Yaskawa INFORM job: X2_50&56A(90,0).JBI

/JOB
//NAME X2_50&56A(90,0)
//POS
///NPOS 390,390,390,18,0,0
///TOOL 0
///POSTYPE PULSE
///PULSE
C00000=-35013,-75230,-81678,-29902,96544,59223
C00001=-146238,44864,29954,-30461,95448,60806
C00002=-147931,42899,30637,-30414,93594,60637
C00003=-149034,42975,32803,-30382,92069,60611
C00004=-149034,43187,33728,-30365,91671,60717
C00005=-148618,42187,30995,-30400,92836,60570
C00006=-146730,40288,31403,-30303,92453,61410
C00007=-147687,41392,32561,-30326,91981,61161
C00008=-146730,40288,31403,-30303,92453,61410
C00009=-146628,38101,29073,-30312,92759,61369
C00010=-146969,35065,25949,-30338,92951,61185
C00011=-146628,38101,29073,-30312,92759,61369
C00012=-145936,38825,28710,-30317,93527,61436
C00013=-144232,40818,28013,-30345,95405,61605
C00014=-133297,17715,2025,-3580,100928,70099
C00015=-121777,-29733,-12388,29914,87306,80525
C00016=-120032,-31040,-9886,30121,84762,80532
C00017=-119311,-31474,-8810,30220,83736,80539
C00018=-119316,-30440,-7071,30243,83270,80413
C00019=-119316,-29997,-6042,30262,82917,80320
C00020=-120906,-31495,-8824,30067,84297,80075
C00021=-122289,-30144,-5697,29969,83711,79393
C00022=-122317,-32815,-7460,29979,83470,79319
C00023=-122289,-30144,-5697,29969,83711,79393
C00024=-122735,-29704,-5039,29928,83710,79223
C00025=-121134,-29738,-5062,30101,83147,79686
C00026=-122735,-29704,-5039,29928,83710,79223
C00027=-126540,-28280,-10143,29422,88423,78984
C00028=-68546,9416,10683,17932,104217,63227
C00029=-68516,6763,11888,17759,102202,62934
C00030=-68503,6025,13208,17671,101063,62768
C00031=-68451,6691,14972,17632,100341,62681
C00032=-68503,5773,12452,17696,101383,62816
C00033=-66565,12547,20523,18047,99542,63243
C00034=-65781,10285,18484,18233,99456,63513
C00035=-66565,12547,20523,18047,99542,63243
C00036=-65967,10809,19346,18174,99249,63415
C00037=-66882,8922,17759,17963,99458,63116
C00038=-65967,10809,19346,18174,99249,63415
C00039=-66084,14240,17447,18358,102066,63804
C00040=-115698,-30544,-51433,15731,84190,63390
C00041=-118338,-32636,-46922,7735,73478,10834
C00042=-114067,48339,9442,8727,107260,-37267
C00043=-101651,53791,20065,8419,102302,-33380
C00044=-100782,53794,25900,8285,98661,-33332
C00045=-100318,54126,27705,8251,97683,-33240
C00046=-100315,54082,28901,8233,96933,-33289
C00047=-100318,54126,27705,8251,97683,-33240
C00048=-103340,51772,25926,13303,96601,-33902
C00049=-102638,52333,26542,13275,96399,-33681
C00050=-103340,51772,25926,13303,96601,-33902
C00051=-103881,51441,24204,13355,97556,-33985
C00052=-105240,51372,17279,13610,101889,-33974
C00053=-105263,53169,23809,16124,107359,-67725
C00054=-105263,53098,24698,16066,106796,-67804
C00055=-105263,53109,24538,16076,106896,-67790
C00056=-105080,50164,21304,16137,107318,-67665
C00057=-105202,52155,23020,16124,107309,-67712
C00058=-106286,50684,21405,16057,107747,-68046
C00059=-106213,46871,17829,16087,107966,-67990
C00060=-105813,47115,18093,16117,107853,-67859
C00061=-106213,47152,15738,16242,109344,-67797
C00062=-102863,-18246,-47623,4026,92422,-23125
C00063=-102376,-34818,-59840,10840,84298,-4292
C00064=-100002,-32974,-49147,13806,76787,-3743
C00065=-100270,-30914,-48271,13869,77337,-3774
C00066=-100148,-31724,-49706,13807,77772,-3684
C00067=-99723,-30030,-48565,13661,77867,-3527
C00068=-99723,-30105,-48044,13677,77517,-3566
C00069=-99495,-31680,-49824,13589,77759,-3462
C00070=-97800,-40718,-55675,5005,73967,4597
C00071=-93318,-38382,-52327,94,72702,9054
C00072=-92851,-38032,-52104,-83,72745,9214
C00073=-95045,-39040,-57560,738,75594,8477
C00074=-124861,-15271,-40833,8838,93503,-41842
C00075=-136908,-36114,-55425,10666,93196,-45849
C00076=-135773,-37299,-49208,10462,88689,-45850
C00077=-136921,-36837,-46377,10628,87355,-46351
C00078=-136921,-36755,-44333,10633,86159,-46454
C00079=-136921,-36814,-45592,10627,86891,-46392
C00080=-117319,-40034,-47848,-16199,85186,-41646
C00081=-117335,-39772,-46156,-16213,84312,-41538
C00082=-116208,-39661,-46084,-16390,84550,-41175
C00083=-118605,-39981,-48556,-15987,85383,-42119
C00084=-142194,-34441,-52424,11225,92893,-47663
C00085=-137296,-41112,-44413,7882,96909,-45970
C00086=-121079,-43154,-38901,8183,90890,-40792
C00087=-119046,-42134,-34632,8196,88600,-40245
C00088=-118232,-41637,-32862,8204,87692,-40026
C00089=-118232,-41216,-31330,8206,86972,-40073
C00090=-118232,-41637,-32862,8204,87692,-40026
C00091=-123515,-41178,-31164,13251,87604,-41880
C00092=-122294,-41232,-31198,13272,87397,-41478
C00093=-123515,-41178,-31164,13251,87604,-41880
C00094=-124446,-41576,-32799,13232,88537,-42104
C00095=-126767,-42340,-36726,13193,90889,-42661
C00096=-121202,-54016,-38461,8184,85107,-41211
C00097=-118951,-52355,-33810,8234,82889,-40587
C00098=-118051,-51605,-31888,8256,82008,-40337
C00099=-118051,-50970,-30224,8268,81318,-40383
C00100=-118051,-51605,-31888,8256,82008,-40337
C00101=-123729,-51057,-30474,13322,82279,-42525
C00102=-122379,-51113,-30506,13351,82049,-42081
C00103=-123729,-51057,-30474,13322,82279,-42525
C00104=-120943,-27615,-16514,12405,97908,-68352
C00105=-120948,-30071,-17086,12372,97018,-68441
C00106=-120951,-31730,-18195,12366,96852,-68459
C00107=-120948,-30071,-17086,12372,97018,-68441
C00108=-124760,-51678,-32249,13279,83200,-42783
C00109=-127326,-53005,-36529,13179,85520,-43425
C00110=-154326,-120554,-77654,11334,79888,-63138
C00111=-167720,-105639,-119673,16034,110248,-69380
C00112=-180425,17295,-38776,18903,121217,-77748
C00113=-160704,-72602,-79591,10350,105538,-81389
C00114=-159985,-76902,-77997,10237,102306,-81413
C00115=-158839,-75685,-75597,10284,101324,-81094
C00116=-158717,-75119,-73898,10260,100564,-81114
C00117=-159022,-76399,-75134,10243,100704,-81209
C00118=-159327,-81052,-76621,10164,99289,-81434
C00119=-159429,-77687,-75590,10198,100380,-81379
C00120=-160454,-72036,-78000,10329,104829,-81362
C00121=-122590,-90956,-95479,-6285,107811,-74232
C00122=-122432,-96187,-93928,-6136,104200,-73988
C00123=-122366,-98076,-93201,-6086,102795,-73894
C00124=-122349,-96392,-90986,-6070,102302,-73864
C00125=-122333,-96702,-91360,-6071,102373,-73862
C00126=-121172,-100063,-92157,-5915,101229,-73400
C00127=-122333,-96702,-91360,-6071,102373,-73862
C00128=-116908,-96303,-91435,-5489,103011,-71994
C00129=-118888,-98383,-91954,-5688,102128,-72646
C00130=-116908,-96303,-91435,-5489,103011,-71994
C00131=-117392,-89431,-93773,-5700,107925,-72394
C00132=-123779,-92334,-96085,11860,100478,-68930
C00133=-121799,-96099,-93963,11739,97018,-68578
C00134=-121068,-94931,-92225,11724,96454,-68379
C00135=-120976,-95732,-90808,11689,95182,-68467
C00136=-121047,-96000,-91535,11697,95495,-68462
C00137=-119860,-99344,-92335,11668,94123,-68181
C00138=-121047,-96000,-91535,11697,95495,-68462
C00139=-119543,-98346,-92112,11677,94445,-68041
C00140=-121592,-100306,-92571,11657,94029,-68789
C00141=-119543,-98346,-92112,11677,94445,-68041
C00142=-122418,-93690,-95360,11815,99162,-68586
C00143=-124052,-92327,-98574,11935,102020,-68874
C00144=-122075,-96496,-96608,11789,98453,-68536
C00145=-121256,-97943,-95721,11744,97072,-68385
C00146=-121250,-96320,-93531,11728,96567,-68431
C00147=-121163,-96877,-94234,11732,96698,-68388
C00148=-119974,-100369,-95083,11696,95280,-68111
C00149=-121163,-96877,-94234,11732,96698,-68388
C00150=-120506,-98881,-94746,11711,95903,-68236
C00151=-118500,-96784,-94222,11730,96355,-67499
C00152=-120506,-98881,-94746,11711,95903,-68236
C00153=-123349,-93657,-97773,11879,100767,-68753
C00154=-135291,-86613,-75974,52977,86020,-81582
C00155=-131116,-88371,-74218,52881,82397,-81428
C00156=-129398,-88910,-73439,52861,80942,-81342
C00157=-128447,-91701,-74067,52932,79748,-81525
C00158=-130431,-95374,-76659,53055,80707,-82053
C00159=-128834,-93195,-74891,52983,79809,-81703
C00160=-130431,-95374,-76659,53055,80707,-82053
C00161=-124555,-94103,-78793,52446,78563,-80078
C00162=-125999,-93781,-77341,52659,78933,-80655
C00163=-124555,-94103,-78793,52446,78563,-80078
C00164=-130787,-92210,-81525,52671,83776,-80437
C00165=-125882,-96985,-97972,20817,92084,-56602
C00166=-122325,-98161,-95172,20440,89016,-55857
C00167=-120880,-94284,-92066,20293,88735,-55390
C00168=-120880,-94153,-90803,20292,88068,-55501
C00169=-120880,-94284,-92066,20293,88735,-55390
C00170=-119026,-94251,-92054,20095,88291,-54803
C00171=-120880,-94284,-92066,20293,88735,-55390
C00172=-120884,-98206,-92897,20294,87320,-55628
C00173=-120880,-94284,-92066,20293,88735,-55390
C00174=-125854,-95536,-95978,20803,91624,-56671
C00175=-125850,-66912,-79659,30836,57983,-58657
C00176=-122561,-63207,-75462,29110,56252,-57732
C00177=-121295,-61670,-73737,28426,55590,-57365
C00178=-121291,-60661,-71640,28674,54906,-57565
C00179=-121285,-60765,-71809,28654,54949,-57550
C00180=-119473,-60737,-71796,27523,54360,-56906
C00181=-121285,-60765,-71809,28654,54949,-57550
C00182=-119935,-60692,-71734,27818,54496,-57075
C00183=-119959,-57359,-70502,27528,55354,-56840
C00184=-119935,-60692,-71734,27818,54496,-57075
C00185=-124401,-66105,-77764,30230,56821,-58377
C00186=-128142,-64639,-90036,18676,74706,-62694
C00187=-138485,-71827,-101197,-11106,105399,-77644
C00188=-147024,-87385,-83593,-35439,109592,-87133
C00189=-149732,-92665,-83137,-35225,106008,-87097
C00190=-150982,-92517,-82536,-35527,105093,-87095
C00191=-150854,-90774,-79322,-35312,104257,-86759
C00192=-145431,-93697,-76928,-39294,101207,-75263
C00193=-143884,-94649,-78323,-39224,102144,-74704
C00194=-141496,-90316,-79520,-39399,105550,-74933
C00195=-154875,-73459,-94031,3699,115712,-75473
C00196=-154642,-88430,-80864,46638,100530,-71967
C00197=-150685,-92332,-80273,46535,96810,-71811
C00198=-149068,-93915,-80023,46523,95290,-71747
C00199=-152233,-91403,-76041,46197,96115,-72893
C00200=-138023,-100193,-87798,32403,89280,-71025
C00201=-139486,-99224,-88637,32451,90704,-71199
C00202=-143008,-96307,-90518,32622,94313,-71562
C00203=-126401,-92982,-99947,26116,71912,-46119
C00204=-122401,-89174,-95921,24616,70248,-44972
C00205=-121170,-87691,-94393,24143,69731,-44617
C00206=-121073,-40431,-77118,23973,104037,-41292
C00207=-121948,-141376,-105315,24084,72465,-47862
C00208=-119793,-124223,-100539,21665,86903,-40754
C00209=-121070,-126388,-102412,21638,87354,-41108
C00210=-126026,-127807,-105919,21532,89991,-42436
C00211=-136654,-67846,-101646,-5444,103045,-74682
C00212=-128322,-96725,-99076,14451,99613,-67284
C00213=-128011,-95143,-96681,14417,98917,-67259
C00214=-125059,-98267,-95078,14269,95825,-66574
C00215=-132883,-103944,-96240,14189,95056,-69399
C00216=-122114,-97273,-96139,7492,99903,-69823
C00217=-123656,-92823,-98050,7552,103478,-70135
C00218=-148370,-106244,-91268,32547,97235,-62203
C00219=-143957,-109023,-89633,32719,93465,-61524
C00220=-142187,-110300,-89017,32799,91899,-61269
C00221=-110014,-102343,-95219,10833,94604,-66470
C00222=-122878,-112804,-97097,10537,93258,-71032
C00223=-110561,-104342,-93907,1603,99479,-78541
C00224=-110841,-84726,-85708,1760,111290,-78449
C00225=-111201,-78802,-86432,1737,114786,-78527
C00226=-106717,-60158,-79706,8194,107324,-64031
C00227=-105123,-63987,-78019,8070,104193,-63696
C00228=-104341,-64830,-77125,8038,103145,-63496
C00229=-106614,-68907,-78610,7970,102193,-64341
C00230=-164586,-101102,-83968,4841,93825,-84736
C00231=-168005,-100380,-83271,4564,93970,-85900
C00232=-165984,-96075,-92358,4843,101626,-84914
C00233=-181857,-131319,-116911,12842,90499,-90722
C00234=-202989,-63880,-99903,47799,99542,-84030
C00235=-168472,-147890,-132681,14947,97151,-71352
C00236=-154326,-120554,-77654,11334,79888,-63138
C00237=-128098,-77833,-51544,-1657,63239,-16727
C00238=-116532,-49017,-34945,-4360,90951,-81305
C00239=-116532,-49017,-34945,-4360,90951,-81305
C00240=-116798,-50663,-32111,-4378,88355,-81305
C00241=-116908,-51227,-30905,-4388,87320,-81307
C00242=-119609,-51392,-30999,-4620,87132,-82211
C00243=-121719,-51405,-31006,-4797,87008,-82917
C00244=-124421,-51272,-30929,-5019,86875,-83824
C00245=-124228,-50732,-32149,-5002,87911,-83800
C00246=-145745,-14259,570,10366,107018,-74117
C00247=-149880,-18384,-846,13396,104500,-71178
C00248=-151111,-18464,18,13945,103653,-70648
C00249=-151285,-17723,1623,13844,103092,-70775
C00250=-151490,-18588,-4768,14034,106516,-70446
C00251=-99208,-22167,-7317,-16130,105202,-90552
C00252=-102111,-21459,-2862,-15110,103391,-89386
C00253=-101894,-21074,-1790,-15006,102986,-89257
C00254=-101783,-20670,-1192,-14957,102851,-89201
C00255=-100868,-20755,-6903,-14931,106373,-89315
C00256=-123764,-49143,-35016,-4968,90511,-83746
C00257=-123498,-46334,-32145,14225,106729,-81506
C00258=-122671,-49917,-31274,14287,104276,-81501
C00259=-122321,-51270,-30849,14324,103286,-81493
C00260=-121710,-51281,-30881,14509,103202,-81284
C00261=-119621,-51322,-31009,15133,102879,-80573
C00262=-119011,-51335,-31052,15312,102775,-80367
C00263=-119414,-50002,-31488,15265,103772,-80384
C00264=-116044,-49795,-31370,16241,103155,-79243
C00265=-112158,-52942,-30337,13826,98266,-82965
C00266=-122910,-69671,-38655,20695,87695,-72461
C00267=-124804,-70759,-45426,20434,91550,-72479
C00268=-120368,-46468,-32388,15179,106240,-80415
C00269=-103583,-18395,-21065,18333,98049,-47386
C00270=-95522,-2033,346,19157,86542,-33647
C00271=-95065,-1179,4289,19188,84551,-33796
C00272=-94194,-282,6213,19202,83664,-33623
C00273=-92524,-10041,-1636,19198,83097,-33115
C00274=-94699,28090,37444,23065,99649,-38348
C00275=-95245,43682,55653,23027,103524,-40317
C00276=-97031,45002,54317,22569,105398,-40615
C00277=-95302,21282,15864,17128,100326,-40606
C00278=-95633,-1961,-1285,16168,78923,-31701
C00279=-94125,315,3726,16087,76781,-31446
C00280=-93197,3589,10969,16156,73926,-31495
C00281=-93115,4380,12654,16195,73301,-31552
C00282=-94556,14113,21261,16393,73308,-32073
C00283=-94819,12763,18273,16338,74461,-32010
C00284=-94855,11979,15831,16266,75524,-31879
C00285=-94760,268,4885,16208,76196,-31753
C00286=-93262,3253,10079,16136,74301,-31466
C00287=-93099,4430,12776,16195,73253,-31551
C00288=-94504,14241,21527,16396,73200,-32069
C00289=-94774,13150,19338,16366,74011,-32057
C00290=-95480,10422,13554,16303,76229,-32007
C00291=-97216,11756,13085,16445,77515,-32459
C00292=-95984,14761,19072,16436,75210,-32328
C00293=-95926,15643,20974,16479,74507,-32404
C00294=-96702,21319,26244,16596,74351,-32707
C00295=-88276,-5311,8070,1704,50857,-22867
C00296=-87929,-9523,3732,1524,51354,-22713
C00297=-88057,-15039,-3820,1549,53169,-22739
C00298=-99387,-43194,-40222,6284,61646,-26942
C00299=-121163,30977,-5145,19643,99311,-32181
C00300=-111536,75135,35465,20047,103602,-28019
C00301=-109733,75701,42270,19665,99503,-28062
C00302=-107396,77633,44085,15199,99812,-27662
C00303=-106846,74881,40767,13783,95666,-18812
C00304=-105506,42598,5344,10183,85057,-21764
C00305=-107494,36842,-4476,11925,85901,-22339
C00306=-110038,51949,7342,17956,100045,-24263
C00307=-110492,43774,10982,19918,106123,-35860
C00308=-109482,36992,6821,19832,105013,-35683
C00309=-108373,36531,10179,19621,102581,-35693
C00310=-107789,34301,9135,19587,101968,-35584
C00311=-105866,51618,28942,18605,112563,-37835
C00312=-106064,56056,31872,17240,113701,-37835
C00313=-105930,58571,31891,15493,114477,-37831
C00314=-113418,37409,2332,24084,99798,-37219
C00315=-113418,37409,2332,24084,105102,-80908
C00316=-113160,50873,23237,25434,107555,-80153
C00317=-112025,51272,23640,25519,107174,-79798
C00318=-112126,54336,25481,25581,107605,-79738
C00319=-108217,56173,27527,25805,106134,-78563
C00320=-108012,53365,25864,25757,105690,-78586
C00321=-107358,53539,26056,25793,105464,-78385
C00322=-107594,58308,28543,25913,106367,-78268
C00323=-114507,53473,22978,25568,109314,-80271
C00324=-122054,65837,41057,36395,121722,-57977
C00325=-123579,42738,19822,41051,112959,-51179
C00326=-124152,34164,13148,42323,109003,-48943
C00327=-124227,34353,16593,41799,107514,-49624
C00328=-126462,36438,15351,42046,109959,-49631
C00329=-128176,29859,1512,43519,114603,-48350
C00330=-130467,-18606,-44219,44095,94408,31747
C00331=-121945,-44389,-49110,46115,69080,26022
C00332=-121904,-40131,-44420,46290,68567,25788
C00333=-113124,-39530,-44042,43500,64204,28113
C00334=-112945,-43259,-50161,42865,65486,28791
C00335=-113288,-45265,-40830,46737,56763,24195
C00336=-111978,-45017,-40682,46242,56106,24578
C00337=-111880,-47039,-43845,45778,56697,24958
C00338=-122010,-47932,-44372,49222,61967,22192
C00339=-118733,-49642,-44567,45028,57156,26003
C00340=-115692,-49409,-44472,43850,55672,26913
C00341=-119979,-54076,-53442,44153,60090,26830
C00342=-127641,-46610,-57429,46858,74797,25997
C00343=-135004,-69306,-84470,28637,83306,-48309
C00344=-114761,-54427,-46396,25764,86438,-35617
C00345=-80124,-32108,-24664,-24795,97657,55749
C00346=-97606,39512,4524,-30816,78189,70702
C00347=-104188,47256,24507,-29638,68650,70716
C00348=-105086,62165,41181,-29824,66062,71062
C00349=-101009,53751,26030,-30366,71859,71113
C00350=-95324,41094,10845,-31949,76382,71947
C00351=-87558,21315,-14177,-31275,118027,78587
C00352=-99257,8968,-10542,-28789,118245,76702
C00353=-100154,5822,-7742,-28106,114988,77225
C00354=-99796,6145,-6533,-27877,114593,77484
C00355=-99255,6664,-4734,-27546,114022,77862
C00356=-106453,5544,-9246,-16915,113806,78351
C00357=-106832,8673,-12915,-17628,117423,77625
C00358=-94457,17302,-8508,-14643,121478,81992
C00359=-77268,892,-37386,-36976,90749,74597
C00360=-55933,-105254,-98782,-41109,86932,84870
C00361=-92475,-165326,-103936,3399,48061,-39515
C00362=-111759,-161502,-101201,19707,45151,-81968
C00363=-123409,-143891,-91937,22487,51121,-85856
C00364=-115094,-142630,-90727,15919,48927,-82057
C00365=-105882,-142342,-91359,8372,48357,-77561
C00366=-52718,-102797,-81138,-14928,68501,-56921
C00367=-53797,-105289,-84123,-14624,68845,-57366
C00368=-54179,-107975,-89277,-14378,70514,-57714
C00369=-16825,-139657,-107848,-21320,74237,-44453
C00370=-66236,-90220,-90975,-10827,78579,-62854
C00371=-122101,-64375,-67751,-40173,89594,55761
C00372=-156986,-41604,-45171,-29986,98885,59603
C00373=-155731,-42293,-43943,-29820,98361,60236
C00374=-154929,-43117,-42986,-29687,97756,60706
C00375=-153721,-35903,-42964,-30012,101405,60215
C00376=-179914,1575,-16772,-26098,97627,80362
C00377=-181040,-1205,-15738,-27877,97095,79905
C00378=-186013,24876,7927,-21128,113140,88491
C00379=-185389,33946,13173,-21244,114639,88446
C00380=-177403,26176,-5438,-27159,113944,78074
C00381=-151823,-12518,-42142,-23070,112328,88779
C00382=-152493,18688,-15572,6849,111397,-44347
C00383=-169300,28033,23113,47357,108802,-40725
C00384=-166510,22316,19742,47659,106730,-40342
C00385=-162493,41198,38614,47947,103283,-40040
C00386=-166990,43523,36346,47749,107450,-40218
C00387=-158337,-39190,-60597,-25734,96154,60613
C00388=-88024,-77489,-63701,-13885,76466,23572
C00389=2286,-107682,-96534,-81,71711,101
BC00000=193562,672653,403459
BC00001=322714,672653,244207
BC00002=322714,672653,244207
BC00003=322714,672653,244207
BC00004=322714,672653,244207
BC00005=322714,672653,244207
BC00006=322714,672653,244207
BC00007=322714,672653,244207
BC00008=322714,672653,244207
BC00009=322714,672653,244207
BC00010=322714,672653,244207
BC00011=322714,672653,244207
BC00012=322714,672653,244207
BC00013=322714,672653,244207
BC00014=299557,698496,312809
BC00015=271448,730733,401387
BC00016=271448,730733,401387
BC00017=271448,730733,401387
BC00018=271448,730733,401387
BC00019=271448,730733,401387
BC00020=271448,730733,401387
BC00021=271448,730733,401387
BC00022=271448,730733,401387
BC00023=271448,730733,401387
BC00024=271448,730733,401387
BC00025=271448,730733,401387
BC00026=271448,730733,401387
BC00027=271448,730733,401387
BC00028=268754,755632,371807
BC00029=268754,755632,371807
BC00030=268754,755632,371807
BC00031=268754,755632,371807
BC00032=268754,755632,371807
BC00033=268754,755632,371807
BC00034=268754,755632,371807
BC00035=268754,755632,371807
BC00036=268754,755632,371807
BC00037=268754,755632,371807
BC00038=268754,755632,371807
BC00039=268754,755632,371807
BC00040=294096,747400,255014
BC00041=331554,773383,228063
BC00042=308865,791089,156472
BC00043=308865,791089,156472
BC00044=308865,791089,156472
BC00045=308865,791089,156472
BC00046=308865,791089,156472
BC00047=308865,791089,156472
BC00048=308865,791089,156472
BC00049=308865,791089,156472
BC00050=308865,791089,156472
BC00051=308865,791089,156472
BC00052=308865,791089,156472
BC00053=308867,791088,156470
BC00054=308867,791088,156470
BC00055=308867,791088,156470
BC00056=308867,791088,156470
BC00057=308867,791088,156470
BC00058=308867,791088,156470
BC00059=308867,791088,156470
BC00060=308867,791088,156470
BC00061=308867,791088,156470
BC00062=308867,791088,156470
BC00063=308867,791088,156470
BC00064=308867,791088,156470
BC00065=308867,791088,156470
BC00066=308867,791088,156470
BC00067=308867,791088,156470
BC00068=308867,791088,156470
BC00069=308867,791088,156470
BC00070=308867,791088,156470
BC00071=308867,791088,156470
BC00072=308867,791088,156470
BC00073=308867,791088,156470
BC00074=337877,791089,225751
BC00075=337877,791089,225751
BC00076=337877,791089,225751
BC00077=337877,791089,225751
BC00078=337877,791089,225751
BC00079=337877,791089,225751
BC00080=337877,791089,225751
BC00081=337877,791089,225751
BC00082=337877,791089,225751
BC00083=337877,791089,225751
BC00084=337877,791089,225751
BC00085=371697,791089,306510
BC00086=371697,791089,306510
BC00087=371697,791089,306510
BC00088=371697,791089,306510
BC00089=371697,791089,306510
BC00090=371697,791089,306510
BC00091=371697,791089,306510
BC00092=371697,791089,306510
BC00093=371697,791089,306510
BC00094=371697,791089,306510
BC00095=371697,791089,306510
BC00096=371795,738368,352691
BC00097=371795,738368,352691
BC00098=371795,738368,352691
BC00099=371795,738368,352691
BC00100=371795,738368,352691
BC00101=371795,738368,352691
BC00102=371795,738368,352691
BC00103=371795,738368,352691
BC00104=371795,738368,352691
BC00105=371795,738368,352691
BC00106=371795,738368,352691
BC00107=371795,738368,352691
BC00108=371795,738368,352691
BC00109=371795,738368,352691
BC00110=242077,668687,834616
BC00111=140850,740327,1062676
BC00112=97529,734526,1075229
BC00113=15,778942,1075175
BC00114=15,778942,1075175
BC00115=15,778942,1075175
BC00116=15,778942,1075175
BC00117=15,778942,1075175
BC00118=15,778942,1075175
BC00119=15,778942,1075175
BC00120=15,778942,1075175
BC00121=50996,831966,1075175
BC00122=50996,831966,1075175
BC00123=50996,831966,1075175
BC00124=50996,831966,1075175
BC00125=50996,831966,1075175
BC00126=50996,831966,1075175
BC00127=50996,831966,1075175
BC00128=50996,831966,1075175
BC00129=50996,831966,1075175
BC00130=50996,831966,1075175
BC00131=50996,831966,1075175
BC00132=20422,818467,1075175
BC00133=20422,818467,1075175
BC00134=20422,818467,1075175
BC00135=20422,818467,1075175
BC00136=20422,818467,1075175
BC00137=20422,818467,1075175
BC00138=20422,818467,1075175
BC00139=20422,818467,1075175
BC00140=20422,818467,1075175
BC00141=20422,818467,1075175
BC00142=20422,818467,1075175
BC00143=44125,831479,1075175
BC00144=44125,831479,1075175
BC00145=44125,831479,1075175
BC00146=44125,831479,1075175
BC00147=44125,831479,1075175
BC00148=44125,831479,1075175
BC00149=44125,831479,1075175
BC00150=44125,831479,1075175
BC00151=44125,831479,1075175
BC00152=44125,831479,1075175
BC00153=44125,831479,1075175
BC00154=15,810379,1075175
BC00155=15,810379,1075175
BC00156=15,810379,1075175
BC00157=15,810379,1075175
BC00158=15,810379,1075175
BC00159=15,810379,1075175
BC00160=15,810379,1075175
BC00161=15,810379,1075175
BC00162=15,810379,1075175
BC00163=15,810379,1075175
BC00164=15,810379,1075175
BC00165=34940,822046,1075175
BC00166=34940,822046,1075175
BC00167=34940,822046,1075175
BC00168=34940,822046,1075175
BC00169=34940,822046,1075175
BC00170=34940,822046,1075175
BC00171=34940,822046,1075175
BC00172=34940,822046,1075175
BC00173=34940,822046,1075175
BC00174=34940,822046,1075175
BC00175=29651,809197,1075175
BC00176=29651,809197,1075175
BC00177=29651,809197,1075175
BC00178=29651,809197,1075175
BC00179=29651,809197,1075175
BC00180=29651,809197,1075175
BC00181=29651,809197,1075175
BC00182=29651,809197,1075175
BC00183=29651,809197,1075175
BC00184=29651,809197,1075175
BC00185=29651,809197,1075175
BC00186=45964,818909,1075175
BC00187=91026,845738,1075175
BC00188=128384,867980,1075175
BC00189=128384,867980,1075175
BC00190=128384,867980,1075175
BC00191=128384,867980,1075175
BC00192=128384,867980,1075173
BC00193=128384,867980,1075175
BC00194=128384,867980,1075175
BC00195=82948,844814,1075175
BC00196=34758,820245,1075175
BC00197=34758,820245,1075175
BC00198=34758,820245,1075175
BC00199=34758,820245,1075175
BC00200=34758,820245,1075175
BC00201=34758,820245,1075175
BC00202=34758,820245,1075175
BC00203=32401,853301,1075175
BC00204=32401,853301,1075175
BC00205=32401,853301,1075175
BC00206=32401,853301,1075175
BC00207=32401,853301,1075175
BC00208=32401,853301,1075175
BC00209=32401,853301,1075175
BC00210=32401,853301,1075175
BC00211=83020,840972,1075175
BC00212=56028,838057,1075175
BC00213=56028,838057,1075175
BC00214=56028,838058,1075171
BC00215=56028,838058,1075171
BC00216=56028,838057,1075175
BC00217=56028,838057,1075175
BC00218=32245,836307,1075175
BC00219=32245,836307,1075175
BC00220=32245,836307,1075175
BC00221=32245,836307,1075175
BC00222=32245,836307,1075175
BC00223=32245,836307,1075175
BC00224=32245,836307,1075175
BC00225=32245,836307,1075175
BC00226=15,798656,1075175
BC00227=15,798656,1075175
BC00228=15,798656,1075175
BC00229=15,798656,1075175
BC00230=15,798656,1075175
BC00231=15,798656,1075175
BC00232=15,798656,1075175
BC00233=15,798656,1075175
BC00234=97529,734526,1075229
BC00235=140850,740327,1062676
BC00236=242077,668687,834616
BC00237=311377,732610,477412
BC00238=342839,745642,375630
BC00239=342839,745642,375630
BC00240=342839,745642,375630
BC00241=342839,745642,375630
BC00242=342839,745642,375630
BC00243=342839,745642,375630
BC00244=342839,745642,375630
BC00245=342839,745642,375630
BC00246=342839,745642,375630
BC00247=342839,745642,375630
BC00248=342839,745642,375630
BC00249=342839,745642,375630
BC00250=342839,745642,375630
BC00251=342839,745642,375630
BC00252=342839,745642,375630
BC00253=342839,745642,375630
BC00254=342839,745642,375630
BC00255=342839,745642,375630
BC00256=342839,745642,375630
BC00257=362759,774876,329067
BC00258=362759,774876,329067
BC00259=362759,774876,329067
BC00260=362759,774876,329067
BC00261=362759,774876,329067
BC00262=362759,774876,329067
BC00263=362759,774876,329067
BC00264=362759,774876,329067
BC00265=362759,774876,329067
BC00266=362759,774876,329067
BC00267=362759,774876,329067
BC00268=362759,774876,329067
BC00269=315582,728319,335765
BC00270=294619,707632,338741
BC00271=294619,707632,338741
BC00272=294619,707632,338741
BC00273=294619,707632,338741
BC00274=294619,707632,338741
BC00275=294619,707632,338741
BC00276=294619,707632,338741
BC00277=294619,707632,338741
BC00278=290475,700197,355860
BC00279=290475,700197,355860
BC00280=290475,700197,355860
BC00281=290475,700197,355860
BC00282=290475,700197,355860
BC00283=290475,700197,355860
BC00284=290475,700197,355860
BC00285=290370,728444,354524
BC00286=290370,728444,354524
BC00287=290370,728444,354524
BC00288=290370,728444,354524
BC00289=290370,728444,354524
BC00290=290370,728444,354524
BC00291=293289,742586,341876
BC00292=293289,742586,341876
BC00293=293289,742586,341876
BC00294=293289,742586,341876
BC00295=293289,742586,341876
BC00296=293289,742586,341876
BC00297=293289,742586,341876
BC00298=293289,742586,341876
BC00299=316588,791089,199770
BC00300=317791,786510,66721
BC00301=317791,786510,66721
BC00302=317791,786510,66721
BC00303=317791,786510,66721
BC00304=317791,786510,66721
BC00305=317791,786510,66721
BC00306=317791,786510,66721
BC00307=319630,788186,144957
BC00308=319630,788186,144957
BC00309=319630,788186,144957
BC00310=319630,788186,144957
BC00311=319630,788186,144957
BC00312=319630,788186,144957
BC00313=319630,788186,144957
BC00314=319630,788186,144957
BC00315=319630,788186,144957
BC00316=319630,788186,144957
BC00317=319630,788186,144957
BC00318=319630,788186,144957
BC00319=319630,788186,144957
BC00320=319630,788186,144957
BC00321=319630,788186,144957
BC00322=319630,788186,144957
BC00323=319630,788186,144957
BC00324=319630,788186,144957
BC00325=319630,788186,144957
BC00326=319630,788186,144957
BC00327=319630,788186,144957
BC00328=319630,788186,144957
BC00329=319630,788186,144957
BC00330=319630,788186,144957
BC00331=319630,788186,144957
BC00332=319630,788186,144957
BC00333=319630,788186,144957
BC00334=319630,788186,144957
BC00335=319630,788186,144957
BC00336=319630,788186,144957
BC00337=319630,788186,144957
BC00338=319630,788186,144957
BC00339=319630,788186,144957
BC00340=319630,788186,144957
BC00341=319630,788186,144957
BC00342=319630,788186,144957
BC00343=319630,788186,144957
BC00344=240407,672279,360474
BC00345=396329,672279,360474
BC00346=396329,698529,131321
BC00347=396329,698529,131321
BC00348=396329,698529,131321
BC00349=396329,698529,131321
BC00350=395142,698529,198138
BC00351=395142,698529,198138
BC00352=395142,698529,198138
BC00353=395142,698529,198138
BC00354=395142,698529,198138
BC00355=395142,698529,198138
BC00356=395142,698529,198138
BC00357=395142,698529,198138
BC00358=395142,698529,198138
BC00359=391373,698529,410367
BC00360=391373,668457,410367
BC00361=172235,722311,251809
BC00362=102588,763517,193606
BC00363=102588,763517,193606
BC00364=102588,763517,193606
BC00365=102588,763517,193606
BC00366=102588,763517,193606
BC00367=102588,763517,193606
BC00368=102588,763517,193606
BC00369=102588,763517,193606
BC00370=236840,763517,193606
BC00371=301044,763517,193606
BC00372=301044,763517,193605
BC00373=301044,763517,193605
BC00374=301044,763517,193605
BC00375=301044,763517,193606
BC00376=359263,763517,193606
BC00377=359263,763517,193606
BC00378=359263,763517,193606
BC00379=359263,763517,193606
BC00380=359263,763517,193606
BC00381=359263,763517,193606
BC00382=359263,763517,193606
BC00383=359263,763517,193606
BC00384=359263,763517,193606
BC00385=359263,763517,193606
BC00386=359263,763517,193606
BC00387=359263,763517,193606
BC00388=235206,720748,442830
BC00389=84306,671503,1075229
EC00000=798156,0
EC00001=798156,0
EC00002=798156,0
EC00003=798156,0
EC00004=798156,0
EC00005=798156,0
EC00006=798156,0
EC00007=798156,0
EC00008=798156,0
EC00009=798156,0
EC00010=798156,0
EC00011=798156,0
EC00012=798156,0
EC00013=798156,0
EC00014=798156,0
EC00015=798156,0
EC00016=798156,0
EC00017=798156,0
EC00018=798156,0
EC00019=798156,0
EC00020=798156,0
EC00021=798156,0
EC00022=798156,0
EC00023=798156,0
EC00024=798156,0
EC00025=798156,0
EC00026=798156,0
EC00027=798156,0
EC00028=798156,0
EC00029=798156,0
EC00030=798156,0
EC00031=798156,0
EC00032=798156,0
EC00033=798156,0
EC00034=798156,0
EC00035=798156,0
EC00036=798156,0
EC00037=798156,0
EC00038=798156,0
EC00039=798156,0
EC00040=798156,0
EC00041=798156,0
EC00042=798156,0
EC00043=798156,0
EC00044=798156,0
EC00045=798156,0
EC00046=798156,0
EC00047=798156,0
EC00048=798156,0
EC00049=798156,0
EC00050=798156,0
EC00051=798156,0
EC00052=798156,0
EC00053=798155,0
EC00054=798155,0
EC00055=798155,0
EC00056=798155,0
EC00057=798155,0
EC00058=798155,0
EC00059=798155,0
EC00060=798155,0
EC00061=798155,0
EC00062=798155,0
EC00063=798155,0
EC00064=798155,0
EC00065=798155,0
EC00066=798155,0
EC00067=798155,0
EC00068=798155,0
EC00069=798155,0
EC00070=798155,0
EC00071=798155,0
EC00072=798155,0
EC00073=798155,0
EC00074=798156,0
EC00075=798156,0
EC00076=798156,0
EC00077=798156,0
EC00078=798156,0
EC00079=798156,0
EC00080=798156,0
EC00081=798156,0
EC00082=798156,0
EC00083=798156,0
EC00084=798156,0
EC00085=798156,0
EC00086=798156,0
EC00087=798156,0
EC00088=798156,0
EC00089=798156,0
EC00090=798156,0
EC00091=798156,0
EC00092=798156,0
EC00093=798156,0
EC00094=798156,0
EC00095=798156,0
EC00096=798156,0
EC00097=798156,0
EC00098=798156,0
EC00099=798156,0
EC00100=798156,0
EC00101=798156,0
EC00102=798156,0
EC00103=798156,0
EC00104=798156,0
EC00105=798156,0
EC00106=798156,0
EC00107=798156,0
EC00108=798156,0
EC00109=798156,0
EC00110=860042,0
EC00111=895167,0
EC00112=929003,0
EC00113=975524,0
EC00114=975524,0
EC00115=975524,0
EC00116=975524,0
EC00117=975524,0
EC00118=975524,0
EC00119=975524,0
EC00120=975524,0
EC00121=975524,0
EC00122=975524,0
EC00123=975524,0
EC00124=975524,0
EC00125=975524,0
EC00126=975524,0
EC00127=975524,0
EC00128=975524,0
EC00129=975524,0
EC00130=975524,0
EC00131=975524,0
EC00132=975524,0
EC00133=975524,0
EC00134=975524,0
EC00135=975524,0
EC00136=975524,0
EC00137=975524,0
EC00138=975524,0
EC00139=975524,0
EC00140=975524,0
EC00141=975524,0
EC00142=975524,0
EC00143=975524,0
EC00144=975524,0
EC00145=975524,0
EC00146=975524,0
EC00147=975524,0
EC00148=975524,0
EC00149=975524,0
EC00150=975524,0
EC00151=975524,0
EC00152=975524,0
EC00153=975524,0
EC00154=975524,0
EC00155=975524,0
EC00156=975524,0
EC00157=975524,0
EC00158=975524,0
EC00159=975524,0
EC00160=975524,0
EC00161=975524,0
EC00162=975524,0
EC00163=975524,0
EC00164=975524,0
EC00165=975524,0
EC00166=975524,0
EC00167=975524,0
EC00168=975524,0
EC00169=975524,0
EC00170=975524,0
EC00171=975524,0
EC00172=975524,0
EC00173=975524,0
EC00174=975524,0
EC00175=975524,0
EC00176=975524,0
EC00177=975524,0
EC00178=975524,0
EC00179=975524,0
EC00180=975524,0
EC00181=975524,0
EC00182=975524,0
EC00183=975524,0
EC00184=975524,0
EC00185=975524,0
EC00186=975524,0
EC00187=975524,0
EC00188=975524,0
EC00189=975524,0
EC00190=975524,0
EC00191=975524,0
EC00192=975520,1
EC00193=975524,0
EC00194=975524,0
EC00195=975524,0
EC00196=975524,0
EC00197=975524,0
EC00198=975524,0
EC00199=975524,0
EC00200=975524,0
EC00201=975524,0
EC00202=975524,0
EC00203=975524,0
EC00204=975524,0
EC00205=975524,0
EC00206=975524,0
EC00207=975524,0
EC00208=975524,0
EC00209=975524,0
EC00210=975524,0
EC00211=975524,0
EC00212=975524,0
EC00213=975524,0
EC00214=975522,1
EC00215=975522,1
EC00216=975524,0
EC00217=975524,0
EC00218=975524,0
EC00219=975524,0
EC00220=975524,0
EC00221=975524,0
EC00222=975524,0
EC00223=975524,0
EC00224=975524,0
EC00225=975524,0
EC00226=975524,0
EC00227=975524,0
EC00228=975524,0
EC00229=975524,0
EC00230=975524,0
EC00231=975524,0
EC00232=975524,0
EC00233=975524,0
EC00234=929003,0
EC00235=895167,0
EC00236=860042,0
EC00237=817325,0
EC00238=798156,0
EC00239=798156,0
EC00240=798156,0
EC00241=798156,0
EC00242=798156,0
EC00243=798156,0
EC00244=798156,0
EC00245=798156,0
EC00246=798156,0
EC00247=798156,0
EC00248=798156,0
EC00249=798156,0
EC00250=798156,0
EC00251=798156,0
EC00252=798156,0
EC00253=798156,0
EC00254=798156,0
EC00255=798156,0
EC00256=798156,0
EC00257=798156,0
EC00258=798156,0
EC00259=798156,0
EC00260=798156,0
EC00261=798156,0
EC00262=798156,0
EC00263=798156,0
EC00264=798156,0
EC00265=798156,0
EC00266=798156,0
EC00267=798156,0
EC00268=798156,0
EC00269=798156,0
EC00270=798156,0
EC00271=798156,0
EC00272=798156,0
EC00273=798156,0
EC00274=798156,0
EC00275=798156,0
EC00276=798156,0
EC00277=798156,0
EC00278=798156,0
EC00279=798156,0
EC00280=798156,0
EC00281=798156,0
EC00282=798156,0
EC00283=798156,0
EC00284=798156,0
EC00285=798156,0
EC00286=798156,0
EC00287=798156,0
EC00288=798156,0
EC00289=798156,0
EC00290=798156,0
EC00291=798156,0
EC00292=798156,0
EC00293=798156,0
EC00294=798156,0
EC00295=798156,0
EC00296=798156,0
EC00297=798156,0
EC00298=798156,0
EC00299=798156,0
EC00300=798156,0
EC00301=798156,0
EC00302=798156,0
EC00303=798156,0
EC00304=798156,0
EC00305=798156,0
EC00306=798156,0
EC00307=798156,0
EC00308=798156,0
EC00309=798156,0
EC00310=798156,0
EC00311=798156,0
EC00312=798156,0
EC00313=798156,0
EC00314=798156,0
EC00315=798156,0
EC00316=798156,0
EC00317=798156,0
EC00318=798156,0
EC00319=798156,0
EC00320=798156,0
EC00321=798156,0
EC00322=798156,0
EC00323=798156,0
EC00324=798156,0
EC00325=798156,0
EC00326=798156,0
EC00327=798156,0
EC00328=798156,0
EC00329=798156,0
EC00330=798156,0
EC00331=798156,0
EC00332=798156,0
EC00333=798156,0
EC00334=798156,0
EC00335=798156,0
EC00336=798156,0
EC00337=798156,0
EC00338=798156,0
EC00339=798156,0
EC00340=798156,0
EC00341=798156,0
EC00342=798156,0
EC00343=798156,0
EC00344=798156,0
EC00345=798156,0
EC00346=798156,0
EC00347=798156,0
EC00348=798156,0
EC00349=798156,0
EC00350=798156,0
EC00351=798156,0
EC00352=798156,0
EC00353=798156,0
EC00354=798156,0
EC00355=798156,0
EC00356=798156,0
EC00357=798156,0
EC00358=798156,0
EC00359=798156,0
EC00360=798156,0
EC00361=798156,0
EC00362=798156,0
EC00363=798156,0
EC00364=798156,0
EC00365=798156,0
EC00366=798156,0
EC00367=798156,0
EC00368=798156,0
EC00369=798156,0
EC00370=798156,0
EC00371=798156,0
EC00372=798156,0
EC00373=798156,0
EC00374=798156,0
EC00375=798156,0
EC00376=798156,0
EC00377=798156,0
EC00378=798156,0
EC00379=798156,0
EC00380=798156,0
EC00381=798156,0
EC00382=798156,0
EC00383=798156,0
EC00384=798156,0
EC00385=798156,0
EC00386=798156,0
EC00387=798156,0
EC00388=798156,0
EC00389=798156,0
///POSTYPE BASE
///RECTAN
///RCONF 0,0,0,0,0,0,0,0,0,0,0,0,0,0,0,0,0,0,0,0,0,0,0,0
P00006=0.222,-3.123,-1.508,0.0000,0.0000,0.0000
P00021=-0.225,-6.128,-0.405,0.0000,0.0000,0.0000
P00022=0.222,-3.123,-1.508,0.0000,0.0000,0.0000
P00023=0.143,-0.036,0.682,0.0000,0.0000,0.0000
P00024=0.145,-0.552,1.326,0.0000,0.0000,0.0000
P00025=-2.003,0.006,0.728,0.0000,0.0000,0.0000
P00026=0.562,-0.002,-0.337,0.0000,0.0000,0.0000
P00027=-0.746,0.015,-9.096,0.0000,0.0000,0.0000
P00028=-2.237,-0.018,-7.702,0.0000,0.0000,0.0000
P00029=-2.156,-0.086,-4.681,0.0000,0.0000,0.0000
P00030=5.926,-4.294,-1.390,0.0000,0.0000,0.0000
P00032=1.957,0.503,-7.217,0.0000,0.0000,0.0000
///RCONF 0,0,0,0,1,0,0,0,0,0,0,0,0,0,0,0,0,0,0,0,0,0,0,0
P00033=-0.123,0.612,-5.012,0.0000,0.0000,0.0000
///RCONF 0,0,0,0,0,0,0,0,0,0,0,0,0,0,0,0,0,0,0,0,0,0,0,0
P00034=-0.304,0.773,-2.693,0.0000,0.0000,0.0000
P00060=2.327,-2.514,-2.692,0.0000,0.0000,0.0000
P00061=1.575,-3.405,-0.752,0.0000,0.0000,0.0000
P00063=0.036,-0.654,-3.005,0.0000,0.0000,0.0000
P00099=-0.837,6.343,-3.499,0.0000,0.0000,0.0000
//INST
///DATE 2025/03/24 10:07
///ATTR SC,RW
///GROUP1 RB1,BS1
///GROUP2 ST1
NOP
'X2_50&56A(90,0)
'Down
'Path S3714
SFTOF3D
MOVJ C00000 BC00000 VJ=100.00  +MOVJ EC00000 VJ=100.00
MOVJ C00001 BC00001 VJ=100.00  +MOVJ EC00001 VJ=100.00
MOVL C00002 BC00002 V=800.0  +MOVJ EC00002 VJ=100.00
SMOVL C00003 BC00003 V=166.7  +MOVJ EC00003
SREFP 3 C00004 BC00004  +REFP EC00004
CALL JOB:SEARCH-R1-S13D
SET P034 P006
SFTON3D P034
SMOVL C00005 BC00005 V=166.7  +MOVJ EC00005
SMOVL C00006 BC00006 V=166.7  +MOVJ EC00006
SREFP 3 C00007 BC00007  +REFP EC00007
CALL JOB:SEARCH-R1-S13D
SET P034 P006
SFTON3D P034
SMOVL C00008 BC00008 V=166.7  +MOVJ EC00008
SMOVL C00009 BC00009 V=166.7  +MOVJ EC00009
SREFP 3 C00010 BC00010  +REFP EC00010
CALL JOB:SEARCH-R1-S13D
SET P034 P006
SFTON3D P034
SMOVL C00011 BC00011 V=16.7  +MOVJ EC00011
MOVL C00012 BC00012 V=800.0  +MOVJ EC00012 VJ=100.00
MOVL C00013 BC00013 V=1000.0  +MOVJ EC00013 VJ=100.00
'EndPath S3714
MOVJ C00014 BC00014 VJ=100.00  +MOVJ EC00014 VJ=100.00
'Path S3715
SFTOF3D
MOVJ C00015 BC00015 VJ=100.00  +MOVJ EC00015 VJ=100.00
MOVL C00016 BC00016 V=800.0  +MOVJ EC00016 VJ=100.00
SMOVL C00017 BC00017 V=166.7  +MOVJ EC00017
SMOVL C00018 BC00018 V=166.7  +MOVJ EC00018
SREFP 3 C00019 BC00019  +REFP EC00019
CALL JOB:SEARCH-R1-S13D
SET P033 P006
SFTON3D P033
SMOVL C00020 BC00020 V=333.3  +MOVJ EC00020
SMOVL C00021 BC00021 V=166.7  +MOVJ EC00021
SREFP 3 C00022 BC00022  +REFP EC00022
CALL JOB:SEARCH-R1-S13D
SET P033 P006
SFTON3D P033
SMOVL C00023 BC00023 V=166.7  +MOVJ EC00023
SMOVL C00024 BC00024 V=166.7  +MOVJ EC00024
SREFP 3 C00025 BC00025  +REFP EC00025
CALL JOB:SEARCH-R1-S13D
SET P033 P006
SFTON3D P033
SMOVL C00026 BC00026 V=166.7  +MOVJ EC00026
MOVL C00027 BC00027 V=1000.0  +MOVJ EC00027 VJ=100.00
'EndPath S3715
'Path S3716
SFTOF3D
MOVJ C00028 BC00028 VJ=100.00  +MOVJ EC00028 VJ=100.00
MOVL C00029 BC00029 V=800.0  +MOVJ EC00029 VJ=100.00
SMOVL C00030 BC00030 V=166.7  +MOVJ EC00030
SREFP 3 C00031 BC00031  +REFP EC00031
CALL JOB:SEARCH-R1-S13D
SET P032 P006
SFTON3D P032
SMOVL C00032 BC00032 V=166.7  +MOVJ EC00032
SMOVL C00033 BC00033 V=166.7  +MOVJ EC00033
SREFP 3 C00034 BC00034  +REFP EC00034
CALL JOB:SEARCH-R1-S13D
SET P032 P006
SFTON3D P032
SMOVL C00035 BC00035 V=166.7  +MOVJ EC00035
SMOVL C00036 BC00036 V=166.7  +MOVJ EC00036
SREFP 3 C00037 BC00037  +REFP EC00037
CALL JOB:SEARCH-R1-S13D
SET P032 P006
SFTON3D P032
SMOVL C00038 BC00038 V=166.7  +MOVJ EC00038
MOVL C00039 BC00039 V=1000.0  +MOVJ EC00039 VJ=100.00
'EndPath S3716
MOVJ C00040 BC00040 VJ=100.00  +MOVJ EC00040 VJ=100.00
'Path S3717
SFTOF3D
MOVJ C00041 BC00041 VJ=100.00  +MOVJ EC00041 VJ=100.00
MOVJ C00042 BC00042 VJ=100.00  +MOVJ EC00042 VJ=100.00
'Path S4334
SFTOF3D
MOVJ C00043 BC00043 VJ=100.00  +MOVJ EC00043 VJ=100.00
MOVL C00044 BC00044 V=800.0  +MOVJ EC00044 VJ=100.00
SMOVL C00045 BC00045 V=166.7  +MOVJ EC00045
SREFP 3 C00046 BC00046  +REFP EC00046
CALL JOB:SEARCH-R1-S13D
SET P029 P006
SFTON3D P029
SMOVL C00047 BC00047 V=166.7  +MOVJ EC00047
SMOVL C00048 BC00048 V=166.7  +MOVJ EC00048
SREFP 3 C00049 BC00049  +REFP EC00049
CALL JOB:SEARCH-R1-S13D
SET P029 P006
SFTON3D P029
SMOVL C00050 BC00050 V=166.7  +MOVJ EC00050
MOVL C00051 BC00051 V=800.0  +MOVJ EC00051 VJ=100.00
MOVL C00052 BC00052 V=1000.0  +MOVJ EC00052 VJ=100.00
SFTOF3D
SMOVL C00053 BC00053 V=166.7  +MOVJ EC00053
SREFP 3 C00054 BC00054  +REFP EC00054
CALL JOB:SEARCH-R1-S13D
SET P060 P006
SFTON3D P060
SMOVL C00055 BC00055 V=166.7  +MOVJ EC00055
SREFP 3 C00056 BC00056  +REFP EC00056
CALL JOB:SEARCH-R1-S13D
SET P060 P006
SFTON3D P060
SMOVL C00057 BC00057 V=166.7  +MOVJ EC00057
SMOVL C00058 BC00058 V=166.7  +MOVJ EC00058
SMOVL C00059 BC00059 V=166.7  +MOVJ EC00059
SREFP 3 C00060 BC00060  +REFP EC00060
CALL JOB:SEARCH-R1-S13D
SET P060 P006
SFTON3D P060
SMOVL C00061 BC00061 V=166.7  +MOVJ EC00061
SFTOF3D
'POPAWIC SERCH
SMOVL C00062 BC00062 V=166.7  +MOVJ EC00062
SMOVL C00063 BC00063 V=250.0  +MOVJ EC00063
SMOVL C00064 BC00064 V=250.0  +MOVJ EC00064
SREFP 3 C00065 BC00065  +REFP EC00065
CALL JOB:SEARCH-R1-S13D
SET P061 P006
SFTON3D P061
SMOVL C00066 BC00066 V=166.7  +MOVJ EC00066
SMOVL C00067 BC00067 V=166.7  +MOVJ EC00067
SREFP 3 C00068 BC00068  +REFP EC00068
CALL JOB:SEARCH-R1-S13D
SET P061 P006
SFTON3D P061
SMOVL C00069 BC00069 V=166.7  +MOVJ EC00069
SMOVL C00070 BC00070 V=333.3  +MOVJ EC00070
SMOVL C00071 BC00071 V=250.0  +MOVJ EC00071
SREFP 3 C00072 BC00072  +REFP EC00072
CALL JOB:SEARCH-R1-S13D
SET P061 P006
SFTON3D P061
SMOVL C00073 BC00073 V=333.3  +MOVJ EC00073
SFTOF3D
'EndPath S4334
MOVJ C00074 BC00074 VJ=100.00  +MOVJ EC00074 VJ=100.00
MOVJ C00075 BC00075 VJ=100.00  +MOVJ EC00075 VJ=100.00
MOVJ C00076 BC00076 VJ=100.00  +MOVJ EC00076 VJ=100.00
SMOVL C00077 BC00077 V=150.0  +MOVJ EC00077
SREFP 3 C00078 BC00078  +REFP EC00078
CALL JOB:SEARCH-R1-S13D
SET P099 P006
SFTON3D P099
SMOVL C00079 BC00079 V=166.7  +MOVJ EC00079
SMOVL C00080 BC00080 V=250.0  +MOVJ EC00080
SMOVL C00081 BC00081 V=166.7  +MOVJ EC00081
SREFP 3 C00082 BC00082  +REFP EC00082
CALL JOB:SEARCH-R1-S13D
SET P099 P006
SFTON3D P099
SMOVL C00083 BC00083 V=250.0  +MOVJ EC00083
MOVJ C00084 BC00084 VJ=100.00  +MOVJ EC00084 VJ=100.00
MOVJ C00085 BC00085 VJ=100.00  +MOVJ EC00085 VJ=100.00
'Path S4335
SFTOF3D
MOVJ C00086 BC00086 VJ=100.00  +MOVJ EC00086 VJ=100.00
MOVL C00087 BC00087 V=800.0  +MOVJ EC00087 VJ=100.00
SMOVL C00088 BC00088 V=166.7  +MOVJ EC00088
SREFP 3 C00089 BC00089  +REFP EC00089
CALL JOB:SEARCH-R1-S13D
SET P028 P006
SFTON3D P028
SMOVL C00090 BC00090 V=166.7  +MOVJ EC00090
SMOVL C00091 BC00091 V=166.7  +MOVJ EC00091
SREFP 3 C00092 BC00092  +REFP EC00092
CALL JOB:SEARCH-R1-S13D
SET P028 P006
SFTON3D P028
SMOVL C00093 BC00093 V=166.7  +MOVJ EC00093
MOVL C00094 BC00094 V=800.0  +MOVJ EC00094 VJ=100.00
MOVL C00095 BC00095 V=1000.0  +MOVJ EC00095 VJ=100.00
'EndPath S4335
'Path S4336
SFTOF3D
MOVJ C00096 BC00096 VJ=100.00  +MOVJ EC00096 VJ=100.00
MOVL C00097 BC00097 V=800.0  +MOVJ EC00097 VJ=100.00
SMOVL C00098 BC00098 V=166.7  +MOVJ EC00098
SREFP 3 C00099 BC00099  +REFP EC00099
CALL JOB:SEARCH-R1-S13D
SET P027 P006
SFTON3D P027
SMOVL C00100 BC00100 V=166.7  +MOVJ EC00100
SMOVL C00101 BC00101 V=166.7  +MOVJ EC00101
SREFP 3 C00102 BC00102  +REFP EC00102
CALL JOB:SEARCH-R1-S13D
SET P027 P006
SFTON3D P027
SMOVL C00103 BC00103 V=166.7  +MOVJ EC00103
SMOVL C00104 BC00104 V=250.0  +MOVJ EC00104
SMOVL C00105 BC00105 V=166.7  +MOVJ EC00105
SREFP 3 C00106 BC00106  +REFP EC00106
CALL JOB:SEARCH-R1-S13D
SET P027 P006
SFTON3D P027
SMOVL C00107 BC00107 V=166.7  +MOVJ EC00107
SFTOF3D
MOVL C00108 BC00108 V=800.0  +MOVJ EC00108 VJ=100.00
MOVL C00109 BC00109 V=1000.0  +MOVJ EC00109 VJ=100.00
'EndPath S4336
'Up
MOVJ C00110 BC00110 VJ=100.00  +MOVJ EC00110 VJ=100.00
MOVJ C00111 BC00111 VJ=100.00  +MOVJ EC00111 VJ=100.00
MOVJ C00112 BC00112 VJ=100.00  +MOVJ EC00112 VJ=100.00
'Path S3719
SFTOF3D
MOVJ C00113 BC00113 VJ=100.00  +MOVJ EC00113 VJ=100.00
MOVL C00114 BC00114 V=800.0  +MOVJ EC00114 VJ=100.00
SMOVL C00115 BC00115 V=166.7  +MOVJ EC00115
SREFP 3 C00116 BC00116  +REFP EC00116
CALL JOB:SEARCH-R1-S13D
SET P026 P006
SFTON3D P026
SMOVL C00117 BC00117 V=166.7  +MOVJ EC00117
SREFP 3 C00118 BC00118  +REFP EC00118
CALL JOB:SEARCH-R1-S13D
SET P026 P006
SFTON3D P026
SMOVL C00119 BC00119 V=166.7  +MOVJ EC00119
MOVL C00120 BC00120 V=1000.0  +MOVJ EC00120 VJ=100.00
'EndPath S3719
'Path S4337
SFTOF3D
MOVJ C00121 BC00121 VJ=100.00  +MOVJ EC00121 VJ=100.00
MOVL C00122 BC00122 V=800.0  +MOVJ EC00122 VJ=100.00
SMOVL C00123 BC00123 V=166.7  +MOVJ EC00123
SREFP 3 C00124 BC00124  +REFP EC00124
CALL JOB:SEARCH-R1-S13D
SET P025 P006
SFTON3D P025
SMOVL C00125 BC00125 V=166.7  +MOVJ EC00125
SREFP 3 C00126 BC00126  +REFP EC00126
CALL JOB:SEARCH-R1-S13D
SET P025 P006
SFTON3D P025
SMOVL C00127 BC00127 V=166.7  +MOVJ EC00127
SMOVL C00128 BC00128 V=166.7  +MOVJ EC00128
SREFP 3 C00129 BC00129  +REFP EC00129
CALL JOB:SEARCH-R1-S13D
SET P025 P006
SFTON3D P025
SMOVL C00130 BC00130 V=166.7  +MOVJ EC00130
MOVL C00131 BC00131 V=1000.0  +MOVJ EC00131 VJ=100.00
'EndPath S4337
'Path S4338
SFTOF3D
MOVJ C00132 BC00132 VJ=100.00  +MOVJ EC00132 VJ=100.00
MOVL C00133 BC00133 V=800.0  +MOVJ EC00133 VJ=100.00
SMOVL C00134 BC00134 V=166.7  +MOVJ EC00134
SREFP 3 C00135 BC00135  +REFP EC00135
CALL JOB:SEARCH-R1-S13D
SET P024 P006
SFTON3D P024
SMOVL C00136 BC00136 V=166.7  +MOVJ EC00136
SREFP 3 C00137 BC00137  +REFP EC00137
CALL JOB:SEARCH-R1-S13D
SET P024 P006
SFTON3D P024
SMOVL C00138 BC00138 V=166.7  +MOVJ EC00138
SMOVL C00139 BC00139 V=166.7  +MOVJ EC00139
SREFP 3 C00140 BC00140  +REFP EC00140
CALL JOB:SEARCH-R1-S13D
SET P024 P006
SFTON3D P024
SMOVL C00141 BC00141 V=166.7  +MOVJ EC00141
MOVL C00142 BC00142 V=1000.0  +MOVJ EC00142 VJ=100.00
'EndPath S4338
'Path S3720
SFTOF3D
MOVJ C00143 BC00143 VJ=100.00  +MOVJ EC00143 VJ=100.00
MOVL C00144 BC00144 V=800.0  +MOVJ EC00144 VJ=100.00
SMOVL C00145 BC00145 V=166.7  +MOVJ EC00145
SREFP 3 C00146 BC00146  +REFP EC00146
CALL JOB:SEARCH-R1-S13D
SET P023 P006
SFTON3D P023
SMOVL C00147 BC00147 V=166.7  +MOVJ EC00147
SREFP 3 C00148 BC00148  +REFP EC00148
CALL JOB:SEARCH-R1-S13D
SET P023 P006
SFTON3D P023
SMOVL C00149 BC00149 V=166.7  +MOVJ EC00149
SMOVL C00150 BC00150 V=166.7  +MOVJ EC00150
SREFP 3 C00151 BC00151  +REFP EC00151
CALL JOB:SEARCH-R1-S13D
SET P023 P006
SFTON3D P023
SMOVL C00152 BC00152 V=166.7  +MOVJ EC00152
MOVL C00153 BC00153 V=1000.0  +MOVJ EC00153 VJ=100.00
'EndPath S3720
'Path S4726
SFTOF3D
MOVJ C00154 BC00154 VJ=100.00  +MOVJ EC00154 VJ=100.00
MOVL C00155 BC00155 V=800.0  +MOVJ EC00155 VJ=100.00
SMOVL C00156 BC00156 V=166.7  +MOVJ EC00156
SREFP 3 C00157 BC00157  +REFP EC00157
CALL JOB:SEARCH-R1-S13D
SET P063 P006
SFTON3D P063
SMOVL C00158 BC00158 V=166.7  +MOVJ EC00158
SREFP 3 C00159 BC00159  +REFP EC00159
CALL JOB:SEARCH-R1-S13D
SET P063 P006
SFTON3D P063
SMOVL C00160 BC00160 V=166.7  +MOVJ EC00160
SMOVL C00161 BC00161 V=166.7  +MOVJ EC00161
SREFP 3 C00162 BC00162  +REFP EC00162
CALL JOB:SEARCH-R1-S13D
SET P063 P006
SFTON3D P063
SMOVL C00163 BC00163 V=166.7  +MOVJ EC00163
MOVL C00164 BC00164 V=1000.0  +MOVJ EC00164 VJ=100.00
'EndPath S4726
'Path S3721
SFTOF3D
MOVJ C00165 BC00165 VJ=100.00  +MOVJ EC00165 VJ=100.00
MOVL C00166 BC00166 V=800.0  +MOVJ EC00166 VJ=100.00
SMOVL C00167 BC00167 V=166.7  +MOVJ EC00167
SREFP 3 C00168 BC00168  +REFP EC00168
CALL JOB:SEARCH-R1-S13D
SET P022 P006
SFTON3D P022
SMOVL C00169 BC00169 V=166.7  +MOVJ EC00169
SREFP 3 C00170 BC00170  +REFP EC00170
CALL JOB:SEARCH-R1-S13D
SET P022 P006
SFTON3D P022
SMOVL C00171 BC00171 V=166.7  +MOVJ EC00171
SREFP 3 C00172 BC00172  +REFP EC00172
CALL JOB:SEARCH-R1-S13D
SET P022 P006
SFTON3D P022
SMOVL C00173 BC00173 V=166.7  +MOVJ EC00173
MOVL C00174 BC00174 V=1000.0  +MOVJ EC00174 VJ=100.00
'EndPath S3721
'Path S3722
SFTOF3D
MOVJ C00175 BC00175 VJ=100.00  +MOVJ EC00175 VJ=100.00
MOVL C00176 BC00176 V=800.0  +MOVJ EC00176 VJ=100.00
SMOVL C00177 BC00177 V=166.7  +MOVJ EC00177
SREFP 3 C00178 BC00178  +REFP EC00178
CALL JOB:SEARCH-R1-S13D
SET P021 P006
SFTON3D P021
SMOVL C00179 BC00179 V=166.7  +MOVJ EC00179
SREFP 3 C00180 BC00180  +REFP EC00180
CALL JOB:SEARCH-R1-S13D
SET P021 P006
SFTON3D P021
SMOVL C00181 BC00181 V=166.7  +MOVJ EC00181
SMOVL C00182 BC00182 V=166.7  +MOVJ EC00182
SREFP 3 C00183 BC00183  +REFP EC00183
CALL JOB:SEARCH-R1-S13D
SET P021 P006
SFTON3D P021
SMOVL C00184 BC00184 V=166.7  +MOVJ EC00184
MOVL C00185 BC00185 V=1000.0  +MOVJ EC00185 VJ=100.00
'EndPath S3722
MOVJ C00186 BC00186 VJ=100.00  +MOVJ EC00186 VJ=100.00
MOVJ C00187 BC00187 VJ=100.00  +MOVJ EC00187 VJ=100.00
'Path W4727
SFTOF3D
SFTON3D P024
MOVJ C00188 BC00188 VJ=100.00  +MOVJ EC00188 VJ=100.00
SMOVL C00189 BC00189 V=800.0  +MOVJ EC00189
SMOVL C00190 BC00190 V=150.0 PL=0  +MOVJ EC00190
MACRO1 MJ#(0) ARGF14
ARCON
SMOVL C00191 BC00191 V=10.0  +MOVJ EC00191
SMOVL C00192 BC00192 V=10.0  +MOVJ EC00192
ARCOF
SMOVL C00193 BC00193 V=800.0  +MOVJ EC00193
SMOVL C00194 BC00194 V=1000.0  +MOVJ EC00194
SFTOF3D
'EndPath W4727
MOVJ C00195 BC00195 VJ=100.00  +MOVJ EC00195 VJ=100.00
'Path W4728
SFTOF3D
SFTON3D P063
MOVJ C00196 BC00196 VJ=100.00  +MOVJ EC00196 VJ=100.00
SMOVL C00197 BC00197 V=800.0  +MOVJ EC00197
SMOVL C00198 BC00198 V=150.0 PL=0  +MOVJ EC00198
ARCON
SMOVL C00199 BC00199 V=10.0  +MOVJ EC00199
SMOVL C00200 BC00200 V=10.0  +MOVJ EC00200
ARCOF
SMOVL C00201 BC00201 V=800.0  +MOVJ EC00201
SMOVL C00202 BC00202 V=1000.0  +MOVJ EC00202
SFTOF3D
'EndPath W4728
'Path W3723
SFTOF3D
SFTON3D P021
MOVJ C00203 BC00203 VJ=100.00  +MOVJ EC00203 VJ=100.00
SMOVL C00204 BC00204 V=800.0  +MOVJ EC00204
SMOVL C00205 BC00205 V=166.7 PL=0  +MOVJ EC00205
MACRO1 MJ#(0) ARGF9
ARCON
SMOVL C00206 BC00206 V=10.0  +MOVJ EC00206
SFTON3D P022
SMOVL C00207 BC00207 V=10.0  +MOVJ EC00207
SMOVL C00208 BC00208 V=10.0  +MOVJ EC00208
ARCOF
SMOVL C00209 BC00209 V=800.0  +MOVJ EC00209
SMOVL C00210 BC00210 V=1000.0  +MOVJ EC00210
SFTOF3D
'EndPath W3723
MOVJ C00211 BC00211 VJ=100.00  +MOVJ EC00211 VJ=100.00
'Path W3724
SFTOF3D
SFTON3D P022
MOVJ C00212 BC00212 VJ=100.00  +MOVJ EC00212 VJ=100.00
SMOVL C00213 BC00213 V=800.0  +MOVJ EC00213
SMOVL C00214 BC00214 V=166.7 PL=0  +MOVJ EC00214
ARCON
SMOVL C00215 BC00215 V=10.0  +MOVJ EC00215
ARCOF
SMOVL C00216 BC00216 V=800.0  +MOVJ EC00216
SMOVL C00217 BC00217 V=1000.0  +MOVJ EC00217
SFTOF3D
'EndPath W3724
'Path W3725
SFTOF3D
SFTON3D P023
MOVJ C00218 BC00218 VJ=100.00  +MOVJ EC00218 VJ=100.00
SMOVL C00219 BC00219 V=800.0  +MOVJ EC00219
SMOVL C00220 BC00220 V=166.7 PL=0  +MOVJ EC00220
ARCON
SWVON WEV#(60)
SMOVL C00221 BC00221 V=7.5  +MOVJ EC00221
SFTON3D P024
SMOVL C00222 BC00222 V=7.5  +MOVJ EC00222
SMOVL C00223 BC00223 V=7.5  +MOVJ EC00223
ARCOF
SWVOF
SMOVL C00224 BC00224 V=800.0  +MOVJ EC00224
SMOVL C00225 BC00225 V=1000.0  +MOVJ EC00225
SFTOF3D
'EndPath W3725
'Path W3726
SFTOF3D
SFTON3D P025
MOVJ C00226 BC00226 VJ=100.00  +MOVJ EC00226 VJ=100.00
SMOVL C00227 BC00227 V=800.0  +MOVJ EC00227
SMOVL C00228 BC00228 V=166.7 PL=0  +MOVJ EC00228
ARCON
SMOVL C00229 BC00229 V=10.0  +MOVJ EC00229
SFTON3D P026
SMOVL C00230 BC00230 V=10.0  +MOVJ EC00230
SMOVL C00231 BC00231 V=10.0  +MOVJ EC00231
ARCOF
SMOVL C00232 BC00232 V=800.0  +MOVJ EC00232
SMOVL C00233 BC00233 V=1000.0  +MOVJ EC00233
SFTOF3D
'EndPath W3726
'Down
MOVJ C00234 BC00234 VJ=100.00  +MOVJ EC00234 VJ=100.00
MOVJ C00235 BC00235 VJ=100.00  +MOVJ EC00235 VJ=100.00
MOVJ C00236 BC00236 VJ=100.00  +MOVJ EC00236 VJ=100.00
'Path W3727
SFTOF3D
SFTON3D P030
MOVJ C00237 BC00237 VJ=100.00  +MOVJ EC00237 VJ=100.00
MOVJ C00238 BC00238 VJ=100.00  +MOVJ EC00238 VJ=100.00
'Path W3729
SFTOF3D
SFTON3D P033
MOVJ C00239 BC00239 VJ=100.00  +MOVJ EC00239 VJ=100.00
SMOVL C00240 BC00240 V=800.0  +MOVJ EC00240
SMOVL C00241 BC00241 V=166.7 PL=0  +MOVJ EC00241
MACRO1 MJ#(0) ARGF14
ARCON
SMOVL C00242 BC00242 V=10.0  +MOVJ EC00242
SMOVL C00243 BC00243 V=10.0  +MOVJ EC00243
SMOVL C00244 BC00244 V=10.0  +MOVJ EC00244
ARCOF
SMOVL C00245 BC00245 V=800.0  +MOVJ EC00245
SMOVL C00246 BC00246 V=250.0  +MOVJ EC00246
SMOVL C00247 BC00247 V=133.3  +MOVJ EC00247
ARCON
SMOVL C00248 BC00248 V=13.3  +MOVJ EC00248
SMOVL C00249 BC00249 V=13.3  +MOVJ EC00249
ARCOF
SMOVL C00250 BC00250 V=166.7  +MOVJ EC00250
SMOVL C00251 BC00251 V=166.7  +MOVJ EC00251
SMOVL C00252 BC00252 V=166.7 PL=0  +MOVJ EC00252
ARCON
SMOVL C00253 BC00253 V=13.3  +MOVJ EC00253
SMOVL C00254 BC00254 V=13.3  +MOVJ EC00254
ARCOF
SMOVL C00255 BC00255 V=166.7  +MOVJ EC00255
SMOVL C00256 BC00256 V=1000.0  +MOVJ EC00256
SFTOF3D
'EndPath W3729
'Path W3730
SFTOF3D
SFTON3D P032
MOVJ C00257 BC00257 VJ=100.00  +MOVJ EC00257 VJ=100.00
SMOVL C00258 BC00258 V=800.0  +MOVJ EC00258
SMOVL C00259 BC00259 V=166.7 PL=0  +MOVJ EC00259
ARCON
SMOVL C00260 BC00260 V=10.0  +MOVJ EC00260
SMOVL C00261 BC00261 V=11.7  +MOVJ EC00261
SMOVL C00262 BC00262 V=11.7  +MOVJ EC00262
ARCOF
SMOVL C00263 BC00263 V=166.7  +MOVJ EC00263
SMOVL C00264 BC00264 V=166.7  +MOVJ EC00264
MACRO1 MJ#(0) ARGF6
SMOVL C00265 BC00265 V=166.7  +MOVJ EC00265
ARCON
SMOVL C00266 BC00266 V=10.0  +MOVJ EC00266
ARCOF
SMOVL C00267 BC00267 V=166.7  +MOVJ EC00267
SMOVL C00268 BC00268 V=1000.0  +MOVJ EC00268
SFTOF3D
MOVJ C00269 BC00269 VJ=100.00  +MOVJ EC00269 VJ=100.00
'EndPath W3730
'Path W3731
SFTOF3D
SFTON3D P032
SFTOF3D
'EndPath W3731
'Path W4471
SFTOF3D
SFTON3D P027
MOVJ C00270 BC00270 VJ=100.00  +MOVJ EC00270 VJ=100.00
SMOVL C00271 BC00271 V=800.0  +MOVJ EC00271
SMOVL C00272 BC00272 V=150.0 PL=0  +MOVJ EC00272
MACRO1 MJ#(0) ARGF9
ARCON
SMOVL C00273 BC00273 V=10.8  +MOVJ EC00273
SMOVL C00274 BC00274 V=10.8  +MOVJ EC00274
ARCOF
SMOVL C00275 BC00275 V=800.0  +MOVJ EC00275
SMOVL C00276 BC00276 V=1000.0  +MOVJ EC00276
SFTOF3D
'EndPath W4471
MOVJ C00277 BC00277 VJ=100.00  +MOVJ EC00277 VJ=100.00
MOVJ C00278 BC00278 VJ=100.00  +MOVJ EC00278 VJ=100.00
'Path W4472
SFTOF3D
SFTON3D P027
MOVJ C00279 BC00279 VJ=100.00  +MOVJ EC00279 VJ=100.00
SMOVL C00280 BC00280 V=800.0  +MOVJ EC00280
SMOVL C00281 BC00281 V=150.0 PL=0  +MOVJ EC00281
ARCON
SMOVL C00282 BC00282 V=10.8  +MOVJ EC00282
ARCOF
SMOVL C00283 BC00283 V=800.0  +MOVJ EC00283
SMOVL C00284 BC00284 V=1000.0  +MOVJ EC00284
SFTOF3D
'EndPath W4472
'Path W4473
SFTOF3D
SFTON3D P028
MOVJ C00285 BC00285 VJ=100.00  +MOVJ EC00285 VJ=100.00
SMOVL C00286 BC00286 V=800.0  +MOVJ EC00286
SMOVL C00287 BC00287 V=150.0 PL=0  +MOVJ EC00287
ARCON
SMOVL C00288 BC00288 V=10.8  +MOVJ EC00288
ARCOF
SMOVL C00289 BC00289 V=800.0  +MOVJ EC00289
SMOVL C00290 BC00290 V=1000.0  +MOVJ EC00290
SFTOF3D
'EndPath W4473
'Path W4474
SFTOF3D
SFTON3D P028
MOVJ C00291 BC00291 VJ=100.00  +MOVJ EC00291 VJ=100.00
SMOVL C00292 BC00292 V=800.0  +MOVJ EC00292
SMOVL C00293 BC00293 V=150.0 PL=0  +MOVJ EC00293
ARCON
SMOVL C00294 BC00294 V=10.8  +MOVJ EC00294
SMOVL C00295 BC00295 V=10.8  +MOVJ EC00295
ARCOF
SMOVL C00296 BC00296 V=800.0  +MOVJ EC00296
SMOVL C00297 BC00297 V=1000.0  +MOVJ EC00297
SFTOF3D
'EndPath W4474
MOVJ C00298 BC00298 VJ=100.00  +MOVJ EC00298 VJ=100.00
MOVJ C00299 BC00299 VJ=100.00  +MOVJ EC00299 VJ=100.00
'Path W4477
SFTOF3D
SFTON3D P029
MOVJ C00300 BC00300 VJ=100.00  +MOVJ EC00300 VJ=100.00
SMOVL C00301 BC00301 V=800.0  +MOVJ EC00301
SMOVL C00302 BC00302 V=150.0 PL=0  +MOVJ EC00302
ARCON
SMOVL C00303 BC00303 V=10.8  +MOVJ EC00303
ARCOF
SMOVL C00304 BC00304 V=800.0  +MOVJ EC00304
SMOVL C00305 BC00305 V=1000.0  +MOVJ EC00305
SFTOF3D
'EndPath W4477
MOVJ C00306 BC00306 VJ=100.00  +MOVJ EC00306 VJ=100.00
MOVJ C00307 BC00307 VJ=100.00  +MOVJ EC00307 VJ=100.00
'Path W4478
SFTOF3D
SFTON3D P029
MOVJ C00308 BC00308 VJ=100.00  +MOVJ EC00308 VJ=100.00
SMOVL C00309 BC00309 V=800.0  +MOVJ EC00309
SMOVL C00310 BC00310 V=150.0 PL=0  +MOVJ EC00310
ARCON
SMOVL C00311 BC00311 V=10.8  +MOVJ EC00311
ARCOF
SMOVL C00312 BC00312 V=800.0  +MOVJ EC00312
SMOVL C00313 BC00313 V=1000.0  +MOVJ EC00313
SFTOF3D
'EndPath W4478
MOVJ C00314 BC00314 VJ=100.00  +MOVJ EC00314 VJ=100.00
MOVJ C00315 BC00315 VJ=100.00  +MOVJ EC00315 VJ=100.00
SFTON3D P060
MACRO1 MJ#(0) ARGF14
SMOVL C00316 BC00316 V=166.7  +MOVJ EC00316
ARCON
SMOVL C00317 BC00317 V=11.7  +MOVJ EC00317
ARCOF
SMOVL C00318 BC00318 V=133.3  +MOVJ EC00318
SMOVL C00319 BC00319 V=133.3  +MOVJ EC00319
SMOVL C00320 BC00320 V=133.3  +MOVJ EC00320
ARCON
SMOVL C00321 BC00321 V=10.8  +MOVJ EC00321
ARCOF
SMOVL C00322 BC00322 V=333.3  +MOVJ EC00322
MOVJ C00323 BC00323 VJ=100.00  +MOVJ EC00323 VJ=100.00
SFTOF3D
MOVJ C00324 BC00324 VJ=100.00  +MOVJ EC00324 VJ=100.00
MOVJ C00325 BC00325 VJ=100.00  +MOVJ EC00325 VJ=100.00
SFTON3D P061
SMOVL C00326 BC00326 V=133.3  +MOVJ EC00326
ARCON
SMOVL C00327 BC00327 V=11.7  +MOVJ EC00327
ARCOF
SMOVL C00328 BC00328 V=166.7  +MOVJ EC00328
MOVJ C00329 BC00329 VJ=100.00  +MOVJ EC00329 VJ=100.00
MOVJ C00330 BC00330 VJ=100.00  +MOVJ EC00330 VJ=100.00
MOVJ C00331 BC00331 VJ=100.00  +MOVJ EC00331 VJ=100.00
SMOVL C00332 BC00332 V=166.7  +MOVJ EC00332
ARCON
SMOVL C00333 BC00333 V=11.7  +MOVJ EC00333
ARCOF
SMOVL C00334 BC00334 V=133.3  +MOVJ EC00334
SMOVL C00335 BC00335 V=166.7  +MOVJ EC00335
ARCON
SMOVL C00336 BC00336 V=6.7  +MOVJ EC00336
ARCOF
SMOVL C00337 BC00337 V=83.3  +MOVJ EC00337
SMOVL C00338 BC00338 V=166.7  +MOVJ EC00338
SMOVL C00339 BC00339 V=83.3  +MOVJ EC00339
ARCON
SMOVL C00340 BC00340 V=6.7  +MOVJ EC00340
ARCOF
SMOVL C00341 BC00341 V=166.7  +MOVJ EC00341
SFTOF3D
SMOVL C00342 BC00342 V=800.0  +MOVJ EC00342
MOVJ C00343 BC00343 VJ=100.00  +MOVJ EC00343 VJ=100.00
MOVJ C00344 BC00344 VJ=100.00  +MOVJ EC00344 VJ=100.00
MOVJ C00345 BC00345 VJ=100.00  +MOVJ EC00345 VJ=100.00
MOVJ C00346 BC00346 VJ=100.00  +MOVJ EC00346 VJ=100.00
SFTON3D P060
SMOVL C00347 BC00347 V=133.3  +MOVJ EC00347
ARCON
SMOVL C00348 BC00348 V=11.7  +MOVJ EC00348
ARCOF
SMOVL C00349 BC00349 V=250.0  +MOVJ EC00349
SFTOF3D
MOVJ C00350 BC00350 VJ=100.00  +MOVJ EC00350 VJ=100.00
MOVJ C00351 BC00351 VJ=100.00  +MOVJ EC00351 VJ=100.00
MOVJ C00352 BC00352 VJ=100.00  +MOVJ EC00352 VJ=100.00
MACRO1 MJ#(0) ARGF6
SFTON3D P027
SMOVL C00353 BC00353 V=133.3  +MOVJ EC00353
ARCON
SMOVL C00354 BC00354 V=15.0  +MOVJ EC00354
SFTOF3D
SMOVL C00355 BC00355 V=15.0  +MOVJ EC00355
SMOVL C00356 BC00356 V=15.0  +MOVJ EC00356
ARCOF
SMOVL C00357 BC00357 V=166.7  +MOVJ EC00357
SMOVL C00358 BC00358 V=666.7  +MOVJ EC00358
MOVJ C00359 BC00359 VJ=100.00  +MOVJ EC00359 VJ=100.00
MOVJ C00360 BC00360 VJ=100.00  +MOVJ EC00360 VJ=100.00
'Path W3732
SFTOF3D
SFTON3D P034
MOVJ C00361 BC00361 VJ=100.00  +MOVJ EC00361 VJ=100.00
MOVJ C00362 BC00362 VJ=100.00  +MOVJ EC00362 VJ=100.00
SMOVL C00363 BC00363 V=800.0  +MOVJ EC00363
SMOVL C00364 BC00364 V=150.0 PL=0  +MOVJ EC00364
MACRO1 MJ#(0) ARGF14
ARCON
SMOVL C00365 BC00365 V=11.7  +MOVJ EC00365
SMOVL C00366 BC00366 V=11.7  +MOVJ EC00366
ARCOF
SMOVL C00367 BC00367 V=800.0  +MOVJ EC00367
SMOVL C00368 BC00368 V=1000.0  +MOVJ EC00368
MOVJ C00369 BC00369 VJ=100.00  +MOVJ EC00369 VJ=100.00
MOVJ C00370 BC00370 VJ=100.00  +MOVJ EC00370 VJ=100.00
MOVJ C00371 BC00371 VJ=100.00  +MOVJ EC00371 VJ=100.00
SFTON3D P034
SMOVL C00372 BC00372 V=133.3  +MOVJ EC00372
ARCON
SMOVL C00373 BC00373 V=11.7  +MOVJ EC00373
SMOVL C00374 BC00374 V=11.7  +MOVJ EC00374
ARCOF
SMOVL C00375 BC00375 V=166.7  +MOVJ EC00375
SMOVL C00376 BC00376 V=166.7  +MOVJ EC00376
SMOVL C00377 BC00377 V=166.7  +MOVJ EC00377
ARCON
SMOVL C00378 BC00378 V=10.0  +MOVJ EC00378
ARCOF
SMOVL C00379 BC00379 V=133.3  +MOVJ EC00379
SFTOF3D
SMOVL C00380 BC00380 V=333.3  +MOVJ EC00380
MOVJ C00381 BC00381 VJ=100.00  +MOVJ EC00381 VJ=100.00
MOVJ C00382 BC00382 VJ=100.00  +MOVJ EC00382 VJ=100.00
MOVJ C00383 BC00383 VJ=100.00  +MOVJ EC00383 VJ=100.00
SFTON3D P099
SMOVL C00384 BC00384 V=166.7  +MOVJ EC00384
ARCON
SMOVL C00385 BC00385 V=11.7  +MOVJ EC00385
ARCOF
SMOVL C00386 BC00386 V=250.0  +MOVJ EC00386
'EndPath W3732
MOVJ C00387 BC00387 VJ=100.00  +MOVJ EC00387 VJ=100.00
MOVJ C00388 BC00388 VJ=100.00  +MOVJ EC00388 VJ=100.00
MOVJ C00389 BC00389 VJ=100.00  +MOVJ EC00389 VJ=100.00
END
